// TIA Portal V20 export
DATA_BLOCK "ControlNodes"   // DB78
{ DB_Accessible_From_OPC_UA := 'FALSE' }
AUTHOR : ERsystem_FA2_DH. Kim
// stored: DBAccessibleFromOPCUA false, DBAccessibleFromWebserver false, MemoryReserve 100, Namespace Unit1.Em2
   VAR
      em { ExternalWritable := 'False'} : "LAF_typeEmControlNode";
      cm : Struct
         Interlock : Struct
            suctionPadTopUpDown : "LER_typeTwoWayActInterlock";
            suctionPadBtmUpDown : "LER_typeTwoWayActInterlock";
            cutterUpDown : "LER_typeTwoWayActInterlock";
            tapeTopUpDown : "LER_typeTwoWayActInterlock";
            tapeBtmUpDown : "LER_typeTwoWayActInterlock";
            spliceHeadRotateTopFwdBwd : "LER_typeTwoWayActInterlock";
            spliceHeadRotateBtmFwdBwd : "LER_typeTwoWayActInterlock";
            suctionPadTopLeftVaccum : "LER_typeTwoWayActInterlock";
            suctionPadTopRightVaccum : "LER_typeTwoWayActInterlock";
            suctionPadBtmLeftVaccum : "LER_typeTwoWayActInterlock";
            suctionPadBtmRightVaccum : "LER_typeTwoWayActInterlock";
            suctionPadTopTapeVaccum : "LER_typeTwoWayActInterlock";
            suctionPadBtmTapeVaccum : "LER_typeTwoWayActInterlock";
         END_STRUCT;
      END_STRUCT;
      citiMap : "LER_OEM_Data";
      semiAutoSplice : Struct
         jobs : "LAF_typeJobs";
         sequence { S7_SetPoint := 'True'} : "LAF_typeSequence";
         "step" { S7_SetPoint := 'True'} : "LER_typeStep";
         jobInterface : Struct
            requset : Struct
               reqUnwinderTopReWind : Bool;
               reqUnwinderBtmReWind : Bool;
               reqEm0To1LinkChg : Bool;
               reqEm1To0LinkChg : Bool;
               reqDancerOn : Bool;
               reqDancerOff : Bool;
            END_STRUCT;
            ready : Struct
               null : Bool;
            END_STRUCT;
            busy : Struct
               busyAutoSplice : Bool;
            END_STRUCT;
            done : Struct
               doneAutoSplice : Bool;
            END_STRUCT;
            workingDone : Struct
               homeJob1WorkingDone { S7_SetPoint := 'True'} : Bool;
               suctionPadUpJob2WorkingDone : Bool;
               topSepaVaccumJob3WorkingDone : Bool;
               btmSepaVaccumJob4WorkingDone : Bool;
               cuttingJob5WorkingDone : Bool;
               topSepaTransferJob6WorkingDone : Bool;
               btmSepaTransferJob7WorkingDone : Bool;
               suctionPadDownJob8WorkingDone : Bool;
               topSepaReMoveJob9WorkingDone : Bool;
               btmSepaReMoveJob10WorkingDone : Bool;
               topSpliceRoateJob11WorkingDone : Bool;
               btmSpliceRoateJob12WorkingDone : Bool;
               topTapingStartJob13WorkingDone : Bool;
               btmTapingStartJob14WorkingDone : Bool;
               tapingFinishJob15WorkingDone : Bool;
               fullAutoSplicingJob30WorkingDone : Bool;
            END_STRUCT;
         END_STRUCT;
         preOperationCheck : Struct
            home : Bool;
            Bool2 : Bool;
            Bool3 : Bool;
            Bool4 : Bool;
            Bool5 : Bool;
            Bool6 : Bool;
            Bool7 : Bool;
            Bool8 : Bool;
            Bool9 : Bool;
         END_STRUCT;
      END_STRUCT;
      emRelations : Struct
         em0 : Struct
            IsLinked : Bool;
            reqAutoSplice : Bool;
            busyAutoSplice : Bool;
            doneAutoSplice : Bool;
         END_STRUCT;
         em1 : Struct
            IsLinked : Bool;
            reqAutoSplice : Bool;
            busyAutoSplice : Bool;
            doneAutoSplice : Bool;
         END_STRUCT;
         em3 : Struct
            cmStatus : Struct
               dancerRegulator : "LBC_typeTwoWayActuatorControlNodeMonitoring";
               dancerEncoder : "LBC_typeAnalogInputControlNodeMonitoring";
            END_STRUCT;
         END_STRUCT;
      END_STRUCT;
      cmSuctionPadTopUpDown { ExternalAccessible := 'False'; ExternalVisible := 'False'; ExternalWritable := 'False'} : "LBC_typeTwoWayActuatorControlNode";
      cmSuctionPadBtmUpDown { ExternalAccessible := 'False'; ExternalVisible := 'False'; ExternalWritable := 'False'; S7_SetPoint := 'True'} : "LBC_typeTwoWayActuatorControlNode";
      cmCutterUpDown { ExternalAccessible := 'False'; ExternalVisible := 'False'; ExternalWritable := 'False'; S7_SetPoint := 'True'} : "LBC_typeTwoWayActuatorControlNode";
      cmTapeTopUpDown { ExternalAccessible := 'False'; ExternalVisible := 'False'; ExternalWritable := 'False'; S7_SetPoint := 'True'} : "LBC_typeTwoWayActuatorControlNode";
      cmTapeBtmUpDown { ExternalAccessible := 'False'; ExternalVisible := 'False'; ExternalWritable := 'False'; S7_SetPoint := 'True'} : "LBC_typeTwoWayActuatorControlNode";
      cmSpliceHeadRotateTopFwdBwd { ExternalAccessible := 'False'; ExternalVisible := 'False'; ExternalWritable := 'False'; S7_SetPoint := 'True'} : "LBC_typeTwoWayActuatorControlNode";
      cmSpliceHeadRotateBtmFwdBwd { ExternalAccessible := 'False'; ExternalVisible := 'False'; ExternalWritable := 'False'; S7_SetPoint := 'True'} : "LBC_typeTwoWayActuatorControlNode";
      cmSuctionPadTopLeftVaccum { ExternalAccessible := 'False'; ExternalVisible := 'False'; ExternalWritable := 'False'; S7_SetPoint := 'True'} : "LBC_typeTwoWayActuatorControlNode";
      cmSuctionPadTopRightVaccum { ExternalAccessible := 'False'; ExternalVisible := 'False'; ExternalWritable := 'False'; S7_SetPoint := 'True'} : "LBC_typeTwoWayActuatorControlNode";
      cmSuctionPadBtmLeftVaccum { ExternalAccessible := 'False'; ExternalVisible := 'False'; ExternalWritable := 'False'; S7_SetPoint := 'True'} : "LBC_typeTwoWayActuatorControlNode";
      cmSuctionPadBtmRightVaccum { ExternalAccessible := 'False'; ExternalVisible := 'False'; ExternalWritable := 'False'; S7_SetPoint := 'True'} : "LBC_typeTwoWayActuatorControlNode";
      cmSuctionPadTopTapeVaccum { ExternalAccessible := 'False'; ExternalVisible := 'False'; ExternalWritable := 'False'; S7_SetPoint := 'True'} : "LBC_typeTwoWayActuatorControlNode";
      cmSuctionPadBtmTapeVaccum { ExternalAccessible := 'False'; ExternalVisible := 'False'; ExternalWritable := 'False'} : "LBC_typeTwoWayActuatorControlNode";
   END_VAR
BEGIN
   // semiAutoSplice."step".action1[101] : Step[101] : Initial Start
   // semiAutoSplice."step".action1[110] : Step[110] : Cutter Home
   // semiAutoSplice."step".action1[111] : Step[111] : Suction Pad Home
   // semiAutoSplice."step".action1[112] : Step[112] : Tape Pad Home
   // semiAutoSplice."step".action1[113] : Step[113] : Splice Head Rotate Home
   // semiAutoSplice."step".action1[114] : Step[114] : Vaccum Home
   // semiAutoSplice."step".action1[190] : Step[190] : Initial Complete
   // semiAutoSplice."step".action1[201] : Step[201] : Top to Bottom Start
   // semiAutoSplice."step".action1[210] : Step[210] : Top Suction Pad Right Vaccum work
   // semiAutoSplice."step".action1[212] : Step[212] : Suction Pad Top & Bottom Work
   // semiAutoSplice."step".action1[214] : Step[214] : Bottom Suction Pad right Vaccum Work
   // semiAutoSplice."step".action1[216] : Step[216] : Cutting Work
   // semiAutoSplice."step".action1[218] : Step[218] : Cutting Home
   // semiAutoSplice."step".action1[220] : Step[220] : Top Suction Pad right Vaccum Home
   // semiAutoSplice."step".action1[222] : Step[222] : Top Suction Pad Home
   // semiAutoSplice."step".action1[225] : Step[225] : Top Unwinder rewind
   // semiAutoSplice."step".action1[230] : Step[230] : Top Suction Pad Work
   // semiAutoSplice."step".action1[232] : Step[232] : Top Suction Pad Left , Right Vaccum work
   // semiAutoSplice."step".action1[234] : Step[234] : Bottom Suction Pad Left , Right Vaccum Home
   // semiAutoSplice."step".action1[236] : Step[236] : Top Suction Pad Home
   // semiAutoSplice."step".action1[238] : Step[238] : Bottom HEAD ROTATE Work
   // semiAutoSplice."step".action1[240] : Step[240] : Top Suction Pad Work
   // semiAutoSplice."step".action1[242] : Step[242] : Bottom Tapping work
   // semiAutoSplice."step".action1[243] : Step[243] : Bottom Tape Vaccum Home
   // semiAutoSplice."step".action1[247] : Step[247] : Bottom Tapping Home
   // semiAutoSplice."step".action1[249] : Step[249] : Top Suction Pad Left , Right Vaccum Home
   // semiAutoSplice."step".action1[251] : Step[251] : Top Suction Pad Home
   // semiAutoSplice."step".action1[253] : Step[253] : Bottom HEAD ROTATE Home
   // semiAutoSplice."step".action1[255] : Step[255] : Check EPC
   // semiAutoSplice."step".action1[257] : Step[257] : Bottom Suction Pad Home
   // semiAutoSplice."step".action1[290] : Step[290] : Top to Bottom Complete
   // semiAutoSplice."step".action1[301] : Step[301] : btm to Bottom Start
   // semiAutoSplice."step".action1[310] : Step[310] : btm Suction Pad Right Vaccum work
   // semiAutoSplice."step".action1[312] : Step[312] : Suction Pad btm & Bottom Work
   // semiAutoSplice."step".action1[314] : Step[314] : Bottom Suction Pad right Vaccum Work
   // semiAutoSplice."step".action1[316] : Step[316] : Cutting Work
   // semiAutoSplice."step".action1[318] : Step[318] : Cutting Home
   // semiAutoSplice."step".action1[320] : Step[320] : btm Suction Pad right Vaccum Home
   // semiAutoSplice."step".action1[322] : Step[322] : btm Suction Pad Home
   // semiAutoSplice."step".action1[325] : Step[325] : btm Unwinder rewind
   // semiAutoSplice."step".action1[330] : Step[330] : btm Suction Pad Work
   // semiAutoSplice."step".action1[332] : Step[332] : btm Suction Pad Left , Right Vaccum work
   // semiAutoSplice."step".action1[334] : Step[334] : Bottom Suction Pad Left , Right Vaccum Home
   // semiAutoSplice."step".action1[336] : Step[336] : btm Suction Pad Home
   // semiAutoSplice."step".action1[338] : Step[338] : Bottom HEAD ROTATE Work
   // semiAutoSplice."step".action1[340] : Step[340] : btm Suction Pad Work
   // semiAutoSplice."step".action1[342] : Step[342] : Bottom Tapping work
   // semiAutoSplice."step".action1[343] : Step[343] : Bottom Tape Vaccum Home
   // semiAutoSplice."step".action1[347] : Step[347] : Bottom Tapping Home
   // semiAutoSplice."step".action1[349] : Step[349] : btm Suction Pad Left , Right Vaccum Home
   // semiAutoSplice."step".action1[351] : Step[351] : btm Suction Pad Home
   // semiAutoSplice."step".action1[353] : Step[353] : Bottom HEAD ROTATE Home
   // semiAutoSplice."step".action1[355] : Step[355] : Check EPC
   // semiAutoSplice."step".action1[357] : Step[357] : Bottom Suction Pad Home
   // semiAutoSplice."step".action1[390] : Step[390] : btm to Bottom Complete
   // semiAutoSplice."step".transition1[101] : Step[101] : Initial Start
   // semiAutoSplice."step".transition1[110] : Step[110] : Cutter Home
   // semiAutoSplice."step".transition1[111] : Step[111] : Suction Pad Home
   // semiAutoSplice."step".transition1[112] : Step[112] : Tape Pad Home
   // semiAutoSplice."step".transition1[113] : Step[113] : Splice Head Rotate Home
   // semiAutoSplice."step".transition1[114] : Step[114] : Vaccum Home
   // semiAutoSplice."step".transition1[190] : Step[190] : Initial Complete
   // semiAutoSplice."step".transition1[201] : Step[201] : Top to Bottom Start
   // semiAutoSplice."step".transition1[210] : Step[210] : Top Suction Pad Right Vaccum work
   // semiAutoSplice."step".transition1[212] : Step[212] : Suction Pad Top & Bottom Work
   // semiAutoSplice."step".transition1[214] : Step[214] : Bottom Suction Pad right Vaccum Work
   // semiAutoSplice."step".transition1[216] : Step[216] : Cutting Work
   // semiAutoSplice."step".transition1[218] : Step[218] : Cutting Home
   // semiAutoSplice."step".transition1[220] : Step[220] : Top Suction Pad right Vaccum Home
   // semiAutoSplice."step".transition1[222] : Step[222] : Top Suction Pad Home
   // semiAutoSplice."step".transition1[225] : Step[225] : Top Unwinder rewind
   // semiAutoSplice."step".transition1[230] : Step[230] : Top Suction Pad Work
   // semiAutoSplice."step".transition1[232] : Step[232] : Top Suction Pad Left , Right Vaccum work
   // semiAutoSplice."step".transition1[234] : Step[234] : Bottom Suction Pad Left , Right Vaccum Home
   // semiAutoSplice."step".transition1[236] : Step[236] : Top Suction Pad Home
   // semiAutoSplice."step".transition1[238] : Step[238] : Bottom HEAD ROTATE Work
   // semiAutoSplice."step".transition1[240] : Step[240] : Top Suction Pad Work
   // semiAutoSplice."step".transition1[242] : Step[242] : Bottom Tapping work
   // semiAutoSplice."step".transition1[243] : Step[243] : Bottom Tape Vaccum Home
   // semiAutoSplice."step".transition1[247] : Step[247] : Bottom Tapping Home
   // semiAutoSplice."step".transition1[249] : Step[249] : Top Suction Pad Left , Right Vaccum Home
   // semiAutoSplice."step".transition1[251] : Step[251] : Top Suction Pad Home
   // semiAutoSplice."step".transition1[253] : Step[253] : Bottom HEAD ROTATE Home
   // semiAutoSplice."step".transition1[255] : Step[255] : Check EPC
   // semiAutoSplice."step".transition1[257] : Step[257] : Bottom Suction Pad Home
   // semiAutoSplice."step".transition1[290] : Step[290] : Top to Bottom Complete
   // semiAutoSplice."step".transition1[301] : Step[301] : btm to Bottom Start
   // semiAutoSplice."step".transition1[310] : Step[310] : btm Suction Pad Right Vaccum work
   // semiAutoSplice."step".transition1[312] : Step[312] : Suction Pad btm & Bottom Work
   // semiAutoSplice."step".transition1[314] : Step[314] : Bottom Suction Pad right Vaccum Work
   // semiAutoSplice."step".transition1[316] : Step[316] : Cutting Work
   // semiAutoSplice."step".transition1[318] : Step[318] : Cutting Home
   // semiAutoSplice."step".transition1[320] : Step[320] : btm Suction Pad right Vaccum Home
   // semiAutoSplice."step".transition1[322] : Step[322] : btm Suction Pad Home
   // semiAutoSplice."step".transition1[325] : Step[325] : btm Unwinder rewind
   // semiAutoSplice."step".transition1[330] : Step[330] : btm Suction Pad Work
   // semiAutoSplice."step".transition1[332] : Step[332] : btm Suction Pad Left , Right Vaccum work
   // semiAutoSplice."step".transition1[334] : Step[334] : Bottom Suction Pad Left , Right Vaccum Home
   // semiAutoSplice."step".transition1[336] : Step[336] : btm Suction Pad Home
   // semiAutoSplice."step".transition1[338] : Step[338] : Bottom HEAD ROTATE Work
   // semiAutoSplice."step".transition1[340] : Step[340] : btm Suction Pad Work
   // semiAutoSplice."step".transition1[342] : Step[342] : Bottom Tapping work
   // semiAutoSplice."step".transition1[343] : Step[343] : Bottom Tape Vaccum Home
   // semiAutoSplice."step".transition1[347] : Step[347] : Bottom Tapping Home
   // semiAutoSplice."step".transition1[349] : Step[349] : btm Suction Pad Left , Right Vaccum Home
   // semiAutoSplice."step".transition1[351] : Step[351] : btm Suction Pad Home
   // semiAutoSplice."step".transition1[353] : Step[353] : Bottom HEAD ROTATE Home
   // semiAutoSplice."step".transition1[355] : Step[355] : Check EPC
   // semiAutoSplice."step".transition1[357] : Step[357] : Bottom Suction Pad Home
   // semiAutoSplice."step".transition1[390] : Step[390] : btm to Bottom Complete
END_DATA_BLOCK
